% RSLogix 500 project PLC Level 2 Project 8b.RSS, saved by version 8.30.00.16 %
PROJECT "UNTITLED"    % processor: Bul.1763 MicroLogix 1100 Series B %

PROGRAM FILES
  LAD 2 "MAIN"  3 rungs
  LAD 3 "IO CONFIG"  3 rungs
  LAD 4 "CTRL LOGIC"  7 rungs

DATA FILES
  O0 OUTPUT  4 elements
  I1 INPUT  6 elements
  S2 STATUS  66 elements
  B3 BINARY  1 elements
  T4 TIMER  1 elements
  C5 COUNTER  1 elements
  R6 CONTROL  1 elements
  N7 INTEGER  4 elements
  F8 FLOAT  5 elements

LADDER 2 "MAIN"
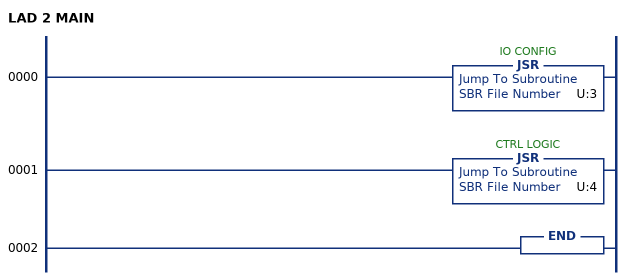
% Rung: 0 %
SOR JSR U:3 EOR
%   U:3  "IO CONFIG" %
% Rung: 1 %
SOR JSR U:4 EOR
%   U:4  "CTRL LOGIC" %
% Rung: 2 %
SOR END EOR

LADDER 3 "IO CONFIG"
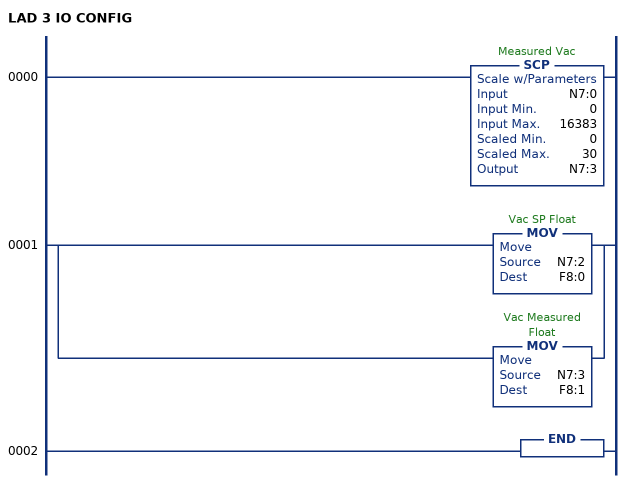
% Rung: 0 %
SOR SCP N7:0 0 16383 0 30 N7:3 EOR
%   N7:0  "Vac sensor in" %
%   N7:3  "Measured Vac" %
% Rung: 1 %
SOR BST MOV N7:2 F8:0 NXB MOV N7:3 F8:1 BND EOR
%   N7:2  "vac SP" %
%   F8:0  "Vac SP Float" %
%   N7:3  "Measured Vac" %
%   F8:1  "Vac Measured Float" %
% Rung: 2 %
SOR END EOR

LADDER 4 "CTRL LOGIC"
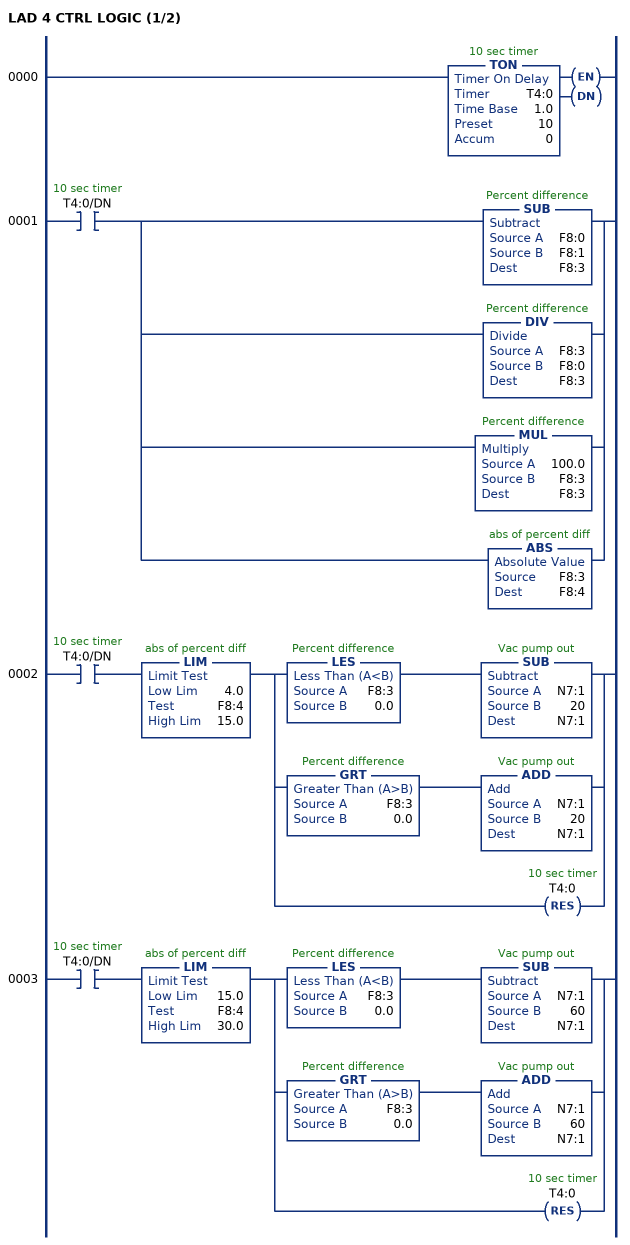
% Rung: 0 %
SOR TON T4:0 1.0 10 0 EOR
%   T4:0  "10 sec timer" %
% Rung: 1 %
SOR XIC T4:0/DN BST SUB F8:0 F8:1 F8:3 NXB DIV F8:3 F8:0 F8:3 NXB MUL 100.0 F8:3 F8:3 NXB ABS F8:3 F8:4 BND EOR
%   T4:0/DN  "10 sec timer" %
%   F8:0  "Vac SP Float" %
%   F8:1  "Vac Measured Float" %
%   F8:3  "Percent difference" %
%   F8:4  "abs of percent diff" %
% Rung: 2 %
SOR XIC T4:0/DN LIM 4.0 F8:4 15.0 BST LES F8:3 0.0 SUB N7:1 20 N7:1 NXB GRT F8:3 0.0 ADD N7:1 20 N7:1 NXB RES T4:0 BND EOR
%   T4:0/DN  "10 sec timer" %
%   F8:4  "abs of percent diff" %
%   F8:3  "Percent difference" %
%   N7:1  "Vac pump out" %
%   T4:0  "10 sec timer" %
% Rung: 3 %
SOR XIC T4:0/DN LIM 15.0 F8:4 30.0 BST LES F8:3 0.0 SUB N7:1 60 N7:1 NXB GRT F8:3 0.0 ADD N7:1 60 N7:1 NXB RES T4:0 BND EOR
%   T4:0/DN  "10 sec timer" %
%   F8:4  "abs of percent diff" %
%   F8:3  "Percent difference" %
%   N7:1  "Vac pump out" %
%   T4:0  "10 sec timer" %

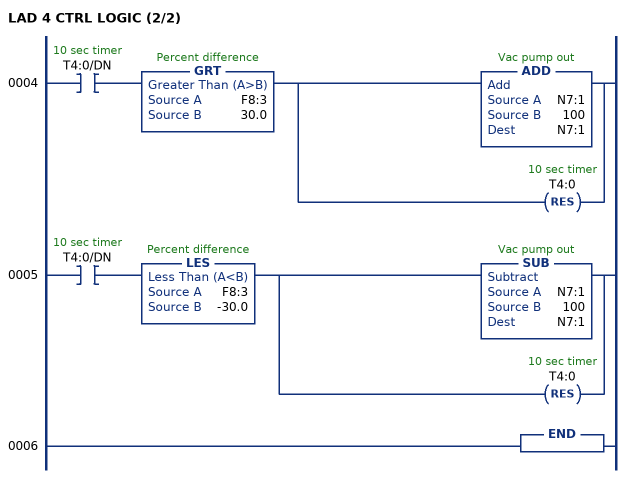
% Rung: 4 %
SOR XIC T4:0/DN GRT F8:3 30.0 BST ADD N7:1 100 N7:1 NXB RES T4:0 BND EOR
%   T4:0/DN  "10 sec timer" %
%   F8:3  "Percent difference" %
%   N7:1  "Vac pump out" %
%   T4:0  "10 sec timer" %
% Rung: 5 %
SOR XIC T4:0/DN LES F8:3 -30.0 BST SUB N7:1 100 N7:1 NXB RES T4:0 BND EOR
%   T4:0/DN  "10 sec timer" %
%   F8:3  "Percent difference" %
%   N7:1  "Vac pump out" %
%   T4:0  "10 sec timer" %
% Rung: 6 %
SOR END EOR

OTHER DOCUMENTED ADDRESSES
  B3:0/0  "Run"
  B3:0/1  "ONS"
  B3:0/2  "Trigger"

DATA TABLE (non-zero values as saved)
DATA T4
% .PRE .ACC %
% T4:0 % 10 0
DATA N7
% N7:0 % 8192 6000 15 0
